// TIA Portal V16 export
// export: Created 2025-12-29T07:35:00.289247Z, ExportSetting WithDefaults, DisplayName Totally Integrated Automation Portal, DisplayVersion V16, DisplayName TIA Portal Version Control Interface, DisplayVersion V16, DisplayName TIA Portal Openness, DisplayVersion V16, DisplayName STEP 7 Professional, DisplayVersion V16, DisplayName STEP 7 Safety, DisplayVersion V16, DisplayName WinCC Professional, DisplayVersion V16
VAR_GLOBAL   // PLC tag table "Tag table from XML_1"
   "Sensor 1" AT %I0.0 : Bool;
   "Pusher 1 front" AT %I0.1 : Bool;
   "Pusher 1 back" AT %I0.2 : Bool;
   "At pusher 1 exit" AT %I0.3 : Bool;
   "Sensor 2" AT %I0.4 : Bool;
   "Pusher 2 front" AT %I0.5 : Bool;
   "Pusher 2 back" AT %I0.6 : Bool;
   "At pusher 2 exit" AT %I0.7 : Bool;
   Start AT %I1.0 : Bool;
   Reset AT %I1.1 : Bool;
   Stop AT %I1.2 : Bool;
   "Emergency stop" AT %I1.3 : Bool;
   "FACTORY I/O (Uruchomiony)" AT %I1.4 : Bool;
   "Entry conveyor 1" AT %Q0.0 : Bool;
   "Pusher 1" AT %Q0.1 : Bool;
   "Conveyor 1" AT %Q0.2 : Bool;
   "Entry conveyor 2" AT %Q0.3 : Bool;
   "Pusher 2" AT %Q0.4 : Bool;
   "Conveyor 2" AT %Q0.5 : Bool;
   "Start light" AT %Q0.6 : Bool;
   "Reset light" AT %Q0.7 : Bool;
   "Stop light" AT %Q1.0 : Bool;
   "Vision sensor 1" AT %ID30 : DInt;
   "Vision sensor 2" AT %ID34 : DInt;
   "Counter 1" AT %QD30 : DInt;
   "Counter 2" AT %QD34 : DInt;
END_VAR
